FUNCTION_BLOCK FB_Discharge
VAR_INPUT
END_VAR
VAR_OUTPUT
END_VAR
VAR
		send_message : PTC_Send_Message;
		fbTimer : TON;
END_VAR

send_message(ID := E_PTC_TX_ID.MAIN_FSM, Command := E_PTC_TX_Command.HV_OFF, CAN_OUTPUts := GVL_PT.CAN_OUTPUTS, CAN_INPUTS := GVL_PT.CAN_INPUTS);

END_FUNCTION_BLOCK

(* stored: Version 1.1.0.1
   POU FB_Discharge: Id {9e10a34e-039c-4453-affc-a15673b4fdc1}, SpecialFunc None *)
